// TwinCAT 3 PLC project PrensaModos
// ProgramVersion: 3.1.4023.0
// libraries:
//   Tc2_MC2, * (Beckhoff Automation GmbH)
//   Tc2_Standard, * (Beckhoff Automation GmbH)
//   Tc2_System, * (Beckhoff Automation GmbH)
//   Tc3_Module, * (Beckhoff Automation GmbH)
//   VisuDialogs, * (System)
//   VisuSymbols,3.5.10.0,System
// project tree:
//   DUTs/ estadosHome.TcDUT, EstadoMando2Manos.TcDUT, EstadosPrensa.TcDUT, Modos.TcDUT
//   / GlobalTextList.TcGTLO, PlcTask.TcTTO, Visualization Manager.TcVMO (not stored)
//   GVLs/ IO.TcGVL, VariablesGlobales.TcGVL
//   POUs/ controlejes.TcPOU, gesAlarmas.TcPOU, MAIN.TcPOU, MandoA2Mans.TcPOU, ModoAutomatico.TcPOU, resetALL.TcPOU, XestionModos.TcPOU
//   VISUs/ SimuladorPrensa.TcVIS
// real-time tasks:
//   TASK PlcTask: cycle T#10ms, priority 20, ADS port 350
// motion (NC):
//   TASK eje1 SAF: cycle T#2ms, priority 4, ADS port 501
//   TASK eje1 SVB: cycle T#10ms, priority 8, ADS port 511
//   AXIS eje1 (id 1)
//     OtherSettings: AllowMotionCmdToSlave=true
//     encoder EncType=1
//     drive DrvType=5
//       Analog: TorqueSetpointScale=10, ScaleFactorActTorque=0.1
//       TimeComp: TaskDelayCycles=1
//     controller CtrType=1
//       CtrPara: PriorControlFactor=1
//         Observer: BandWidth=20
//   AXIS Axis 2 (id 2)
//     OtherSettings: AllowMotionCmdToSlave=true
//     encoder EncType=1
//     drive DrvType=5
//       Analog: TorqueSetpointScale=10, ScaleFactorActTorque=0.1
//       TimeComp: TaskDelayCycles=1
//     controller CtrType=1
//       CtrPara: PriorControlFactor=1
//         Observer: BandWidth=20
// variable links:
//   PrensaModos/PrensaModos Instance <-> eje1 SAF/Axes/Axis 2
//     PlcTask Inputs/VariablesGlobales.eje2.NcToPlc <-> Outputs/ToPlc
//     PlcTask Outputs/VariablesGlobales.eje2.PlcToNc <-> Inputs/FromPlc
//   PrensaModos/PrensaModos Instance <-> eje1 SAF/Axes/eje1
//     PlcTask Inputs/VariablesGlobales.eje1.NcToPlc <-> Outputs/ToPlc
//     PlcTask Outputs/VariablesGlobales.eje1.PlcToNc <-> Inputs/FromPlc

CONFIGURATION PrensaModos
    RESOURCE PLC ON TwinCAT3
        TASK PlcTask(INTERVAL := T#10ms, PRIORITY := 20);
        PROGRAM MAIN WITH PlcTask : MAIN;
    END_RESOURCE
END_CONFIGURATION

// ---- DUTs/estadosHome.TcDUT
{attribute 'qualified_only'}
{attribute 'strict'}
TYPE estadosHome :
(
	subiendo:=0,
	abriendo,
	sacando,
	ok,
	espera
);
END_TYPE

// ---- DUTs/EstadoMando2Manos.TcDUT
{attribute 'qualified_only'}
{attribute 'strict'}
TYPE estadoMando2Manos:
	(
		Esperando:=0,
		Pulsado1,
		Pulsado2,
		Validado,
		Error
	);
END_TYPE

// ---- DUTs/EstadosPrensa.TcDUT
{attribute 'qualified_only'}
{attribute 'strict'}
TYPE EstadosPrensa :
(
	Parada:=0,
	Entrando,
	Pechando,
	Prensando,
	Aguantando,
	Liberando,
	Abrindo,
	Sacando
);
END_TYPE

// ---- DUTs/Modos.TcDUT
{attribute 'qualified_only'}
{attribute 'strict'}
TYPE Modos :
(
	Stop:=0,
	Auto,
	Manual,
	StopSec,
	Reseteando,
	Parando
);
END_TYPE

// ---- GVLs/IO.TcGVL
{attribute 'qualified_only'}
VAR_GLOBAL
	//Entradas modos
	Marcha AT %I*:BOOL;
	Paro AT %I*:BOOL;
	ManualAuto AT %I*:BOOL;
	SafetyOK AT %I*: BOOL;
	ResetErrores AT %I*:BOOL;
	
	//Entradas Modo Manual
	PulsadorEntrar AT %I*:BOOL;
	PulsadorSair AT %I*:BOOL;
	PulsadorPechar AT %I*:BOOL;
	PulsadorAbrir AT %I*:BOOL;
	PulsadorPrensar AT %I*:BOOL;
	PulsadorLiberar AT %I*:BOOL;
	
	//Entradas físicas mando a 2 mans
	Pulsador1 AT %I*: BOOL;
	Pulsador2 AT %I*: BOOL;
END_VAR

// ---- GVLs/VariablesGlobales.TcGVL

VAR_GLOBAL
	ModoMaquina:Modos := modos.StopSec;
	EnErro:BOOL := FALSE;
	Simular:BOOL := TRUE;
	eje1:AXIS_REF; //cinta
	eje2:AXIS_REF; //prensa
	paroAlcanzado: BOOL;
	noFallo: BOOL;
	ErrorEjes: BOOL;
	power1:BOOL:=FALSE;
	power2:BOOL:=FALSE;
	stop1:BOOL:=FALSE;
	stop2:BOOL:=FALSE;
	reset1:BOOL:=FALSE;
	reset2:BOOL:=FALSE;
	mover1:BOOL:=FALSE;
	mover2:BOOL:=FALSE;
	posicion1:UINT:=0;
	posicion2:UINT:=0;
	
END_VAR

// ---- POUs/MAIN.TcPOU
PROGRAM MAIN
VAR
END_VAR

//resetALL();
XestionModos();						//Chamada a Xestión de Modos
MandoA2Mans(LimiteSoster:=NOT modoAutomatico.goHome);	//Chamada o Mando a 2 mans
gesAlarmas();
IF mandoa2mans.Error THEN
	modoautomatico.goHome:=TRUE;
END_IF
//Se estamos en modo automático chamamos o programa
IF VariablesGlobales.ModoMaquina=modos.Auto THEN
	ModoAutomatico(bOrdenMarcha:=MandoA2Mans.Q,
	bSimular:=VariablesGlobales.Simular,
	ordenhome := io.pulsador1);	
END_IF

END_PROGRAM

// ---- POUs/XestionModos.TcPOU
PROGRAM XestionModos
VAR
	fMarcha:r_trig;
	fReset:r_trig;
	
	tResetErros:ton;
END_VAR

fMarcha(clk:=IO.marcha);
fReset(clk:=IO.ResetErrores);
power1:=TRUE;
power2:=TRUE;
stop1:=FALSE;
stop2:=FALSE;

CASE VariablesGlobales.ModoMaquina OF
	modos.Auto:
		IF IO.ManualAuto THEN
			stop1:=TRUE;
			stop2:=TRUE;
			VariablesGlobales.ModoMaquina:=modos.Manual;
		END_IF
		IF IO.Paro THEN
			VariablesGlobales.ModoMaquina:=modos.parando;
		END_IF
		IF VariablesGlobales.EnErro THEN
			VariablesGlobales.ModoMaquina:=modos.StopSec;
		END_IF
	modos.Manual:
		IF NOT IO.ManualAuto THEN
			VariablesGlobales.ModoMaquina:=modos.stop;
		END_IF
		IF VariablesGlobales.EnErro THEN
			VariablesGlobales.ModoMaquina:=modos.StopSec;
		END_IF
	
	modos.Stop:
		IF IO.ManualAuto THEN
			VariablesGlobales.ModoMaquina:=modos.Manual;
		END_IF
		IF fMarcha.q THEN
			VariablesGlobales.ModoMaquina:=modos.Auto;
		END_IF
		IF VariablesGlobales.EnErro THEN
			VariablesGlobales.ModoMaquina:=modos.StopSec;
		END_IF
	
	modos.StopSec:
		power1:=FALSE; //no tiene energía en el stopsec
		power2:=FALSE;
		IF fReset.q THEN
			VariablesGlobales.ModoMaquina:=modos.Reseteando;
			tResetErros(in:=FALSE);
		END_IF
		
	//Temos un novo modo para o reseteo, no que damos medio segundo para que, no caso de haber algunha alarma, esta salte
	modos.Reseteando:
		tResetErros(in:=TRUE, pt:=T#1S);
		IF tResetErros.Q AND NOT EnErro THEN
			VariablesGlobales.ModoMaquina:=modos.Stop;
		END_IF
		//Se o final do temporizador seguimos tendo un erro imos a modo stop seguro
		IF tResetErros.Q AND VariablesGlobales.EnErro THEN
			VariablesGlobales.ModoMaquina:=modos.StopSec;
		END_IF
	modos.Parando:
		stop1:=TRUE;
		stop2:=TRUE;
		IF paroAlcanzado THEN
			VariablesGlobales.ModoMaquina:=modos.Stop;
		END_IF
END_CASE

END_PROGRAM

// ---- POUs/MandoA2Mans.TcPOU
PROGRAM MandoA2Mans
VAR_INPUT
	LimiteSoster:BOOL;
END_VAR
VAR
	flancoP1:r_trig;
	flancoP2:r_trig;
	temp:ton;
	estadoActual:estadoMando2Manos;
END_VAR
VAR_OUTPUT
	Q:BOOL:=FALSE;
	Error:bool:=false;
END_VAR

//Valores por defecto
q:=FALSE;
Error:=FALSE;
//Control de flancos
flancoP1(clk:=IO.Pulsador1 AND ModoAutomatico.EstadoPrensa=EstadosPrensa.Parada);
flancoP2(clk:=IO.Pulsador2 AND ModoAutomatico.EstadoPrensa=EstadosPrensa.Parada);
//Temporizador para detectar a pulsación "simulatanea" dos dous pulsadores
temp(in:=estadoActual=estadoMando2Manos.Pulsado1 OR estadoActual=estadoMando2Manos.Pulsado2, pt:=T#250MS);

CASE estadoActual OF
	estadoMando2Manos.Esperando:
		IF flancoP1.Q THEN
			estadoActual:=estadoMando2Manos.Pulsado1;
		END_IF
		IF flancoP2.Q THEN
			estadoActual:=estadoMando2Manos.Pulsado2;
		END_IF
		IF flancoP1.Q AND flancoP2.Q THEN
			estadoActual:=estadoMando2Manos.Validado;
		END_IF
	estadoMando2Manos.Pulsado1:
		IF temp.Q OR NOT IO.Pulsador1 THEN
			estadoActual:=estadoMando2Manos.Esperando;
		END_IF
		IF flancoP2.Q THEN
			estadoActual:=estadoMando2Manos.Validado;
		END_IF
	estadoMando2Manos.Pulsado2:
		IF temp.Q OR NOT IO.Pulsador2 THEN
			estadoActual:=estadoMando2Manos.Esperando;
		END_IF
		IF flancoP1.Q THEN
			estadoActual:=estadoMando2Manos.Validado;
		END_IF
	estadoMando2Manos.Validado:
		q:=TRUE;
		//Se se cumplen as condicións de límite de mantemento imos a inicio
		IF LimiteSoster THEN
			estadoActual:=estadoMando2Manos.Esperando;
		END_IF
		//Se soltamos algún pulsador imos a erro
		IF NOT io.Pulsador1 OR NOT io.Pulsador2 THEN
			estadoActual:=estadoMando2Manos.Error;
		END_IF
	estadoMando2Manos.Error:
		//Erro estará a TRUE durante un ciclo
		Error:=TRUE;
		estadoActual:=estadoMando2Manos.Esperando;
END_CASE

END_PROGRAM

// ---- POUs/ModoAutomatico.TcPOU
PROGRAM ModoAutomatico
VAR_INPUT
	bOrdenMarcha: BOOL;
	bSimular:BOOL:=TRUE;
	goHome:BOOL := False;
	ordenHome:bool;
END_VAR
VAR_OUTPUT
	bFinCiclo:BOOL :=FALSE;
	EstadoPrensa: EstadosPrensa;
	estadohome: estadoshome;
	
END_VAR
VAR
	//Evolucion
	FlancoMarcha: R_trig;
	TemporizadorPrensado: Ton;
	
	//Simulacion
	TemporizadorSimulacion: TON;
	TempoSimulacion: TIME;
	ForzarErro: BOOL:=FALSE; //Esta variable permitirá forzar un erro de TimeOut
	MC_SetPosition_eje1:mc_setposition;
	MC_SetPosition_eje2:mc_setposition;
END_VAR

IF gohome THEN
	vueltacasa();
END_IF
IF NOT gohome THEN
	EvolucionEstados_Transicions();
	ActivacionActuacions_Lugares();
END_IF
IF bSimular THEN
	SimulacionAutomatico();
	simulacionejes();
END_IF

ACTION ActivacionActuacions_Lugares:
mover1:=FALSE;
mover2:=FALSE;

CASE EstadoPrensa OF
	EstadosPrensa.Entrando:
		posicion1:=1000;
		mover1:=TRUE;
	EstadosPrensa.Prensando:
		posicion2:=1000;
		mover2:=TRUE;
	EstadosPrensa.Liberando:
		posicion2:=0;
		mover2:=TRUE;
	EstadosPrensa.Sacando:
		posicion1:=0;
		mover1:=TRUE;
END_CASE
END_ACTION

ACTION EvolucionEstados_Transicions:
FlancoMarcha(clk:=bOrdenMarcha);
TemporizadorPrensado(in:=EstadoPrensa=EstadosPrensa.Aguantando, PT:=T#3S);
CASE EstadoPrensa OF
	EstadosPrensa.Parada:
		IF flancomarcha.Q THEN
			EstadoPrensa:=EstadosPrensa.Entrando;
		END_IF
	EstadosPrensa.Entrando:
		IF controlejes.MC_MoveAbsolute_eje1.Done THEN
			EstadoPrensa:=EstadosPrensa.Prensando;
		END_IF
	EstadosPrensa.Prensando:
		IF controlejes.MC_MoveAbsolute_eje2.Done THEN
			EstadoPrensa:=EstadosPrensa.Aguantando;
		END_IF
	EstadosPrensa.Aguantando:
		IF TemporizadorPrensado.Q THEN
			EstadoPrensa:=EstadosPrensa.Liberando;
		END_IF
	EstadosPrensa.Liberando:
		IF controlejes.MC_MoveAbsolute_eje1.Done THEN
			EstadoPrensa:=EstadosPrensa.Sacando;
		END_IF
	EstadosPrensa.Sacando:
		IF controlejes.MC_MoveAbsolute_eje1.Done THEN
			EstadoPrensa:=EstadosPrensa.Parada;
			bFinCiclo:=TRUE;
		END_IF
END_CASE
END_ACTION

ACTION SimulacionAutomatico:
//Se estamos simulando o pulsador1 activará ambos pulsadores
io.Pulsador2:=IO.Pulsador1;
TemporizadorSimulacion(IN:=TRUE, PT:=TempoSimulacion);
MC_SetPosition_eje1.execute:=FALSE;
MC_SetPosition_eje2.execute:=FALSE;

CASE EstadoPrensa OF
	EstadosPrensa.Parada:
		TemporizadorSimulacion(IN:=FALSE);
		TempoSimulacion:=T#5S;
		
	EstadosPrensa.Entrando:
		IF TemporizadorSimulacion.Q THEN
			MC_SetPosition_eje1.position:=1000;
			MC_SetPosition_eje1.execute:=TRUE;
			TemporizadorSimulacion(IN:=FALSE);
			TempoSimulacion:=T#2S;
		END_IF
	EstadosPrensa.Prensando:
		IF TemporizadorSimulacion.Q THEN
			MC_SetPosition_eje2.position:=1000;
			MC_SetPosition_eje2.execute:=TRUE;
			TemporizadorSimulacion(IN:=FALSE);
			TempoSimulacion:=T#3S;
		END_IF
	EstadosPrensa.Aguantando:
		TemporizadorSimulacion(IN:=FALSE);
	EstadosPrensa.Liberando:
		IF TemporizadorSimulacion.Q THEN
			MC_SetPosition_eje2.position:=0;
			MC_SetPosition_eje2.execute:=TRUE;
			TemporizadorSimulacion(IN:=FALSE);
			TempoSimulacion:=T#2S;
		END_IF
	EstadosPrensa.Sacando:
		IF TemporizadorSimulacion.Q THEN
			MC_SetPosition_eje1.position:=0;
			MC_SetPosition_eje1.execute:=TRUE;
			TemporizadorSimulacion(IN:=FALSE);
			TempoSimulacion:=T#5S;
		END_IF
END_CASE
//Se queremos forzar un erro metemoslle un minuto o temporizador
IF ForzarErro THEN
	TempoSimulacion:= T#1M;
END_IF
END_ACTION

ACTION simulacionEjes:
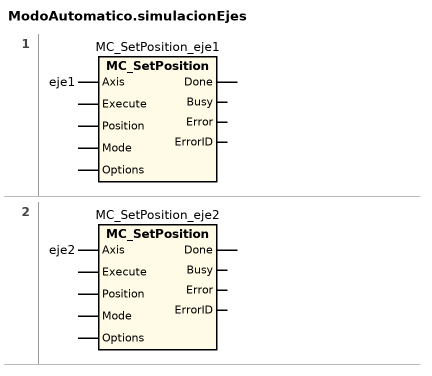
// NETWORK 1
MC_SetPosition_eje1(Axis := eje1); // MC_SetPosition

// NETWORK 2
MC_SetPosition_eje2(Axis := eje2); // MC_SetPosition
END_ACTION

ACTION vueltacasa:
mover1:=FALSE;
mover2:=FALSE;

CASE estadohome OF
	estadoshome.espera:
		IF gohome THEN
			estadohome:= estadoshome.subiendo;
		END_IF
	estadoshome.subiendo:
		posicion2:=0;
		mover2:=TRUE;
		IF controlejes.MC_MoveAbsolute_eje2.Done THEN
			estadohome:= estadoshome.sacando;
		END_IF
	estadoshome.sacando:
		posicion1:=0;
		mover1:=TRUE;
		IF controlejes.MC_MoveAbsolute_eje1.Done THEN
			estadohome:= estadoshome.ok;
		END_IF
	estadoshome.ok:
		estadohome:= estadoshome.espera;
		gohome:=FALSE;
END_CASE
END_ACTION

END_PROGRAM

// ---- POUs/controlejes.TcPOU
PROGRAM controlejes
VAR
	MC_Power_eje1: MC_Power;
	MC_Power_eje2: MC_Power;
	MC_Stop_eje1: mc_stop;
	MC_Stop_eje2: mc_stop;
	MC_Reset_eje1: mc_reset;
	MC_Reset_eje2: mc_reset;
	MC_MoveAbsolute_eje1: MC_MoveAbsolute;
	MC_MoveAbsolute_eje2: MC_MoveAbsolute;
	
	MC_ReadStatus_eje1: MC_ReadStatus;
	MC_ReadStatus_eje2: MC_ReadStatus;
	
	MC_MoveVelocity_0: MC_MoveVelocity;
END_VAR

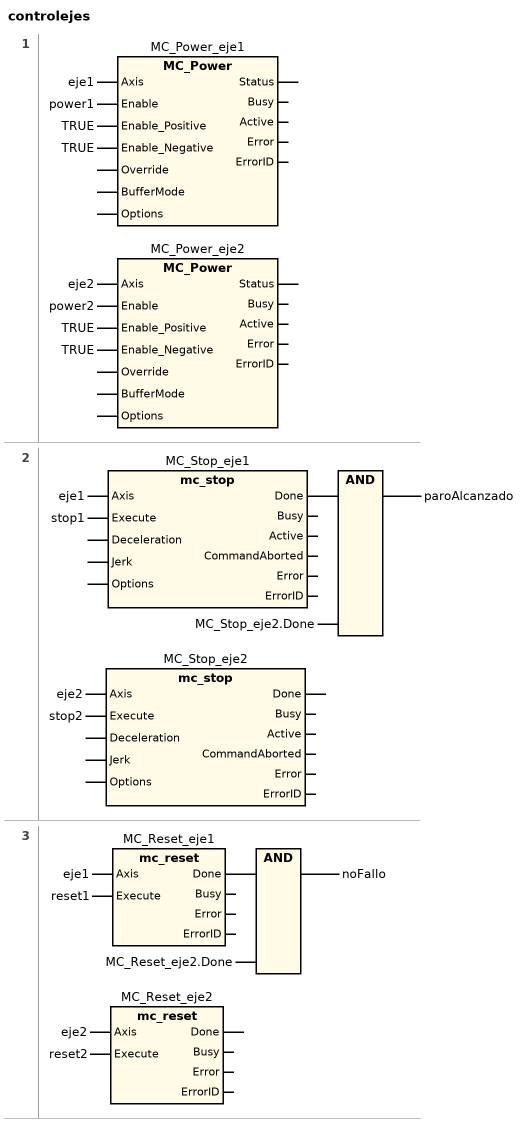
// NETWORK 1
MC_Power_eje1(Axis := eje1, Enable := power1, Enable_Positive := TRUE, Enable_Negative := TRUE); // MC_Power
MC_Power_eje2(Axis := eje2, Enable := power2, Enable_Positive := TRUE, Enable_Negative := TRUE); // MC_Power

// NETWORK 2
MC_Stop_eje1(Axis := eje1, Execute := stop1); // mc_stop
paroAlcanzado := MC_Stop_eje1.Done AND MC_Stop_eje2.Done;
MC_Stop_eje2(Axis := eje2, Execute := stop2); // mc_stop

// NETWORK 3
MC_Reset_eje1(Axis := eje1, Execute := reset1); // mc_reset
noFallo := MC_Reset_eje1.Done AND MC_Reset_eje2.Done;
MC_Reset_eje2(Axis := eje2, Execute := reset2); // mc_reset

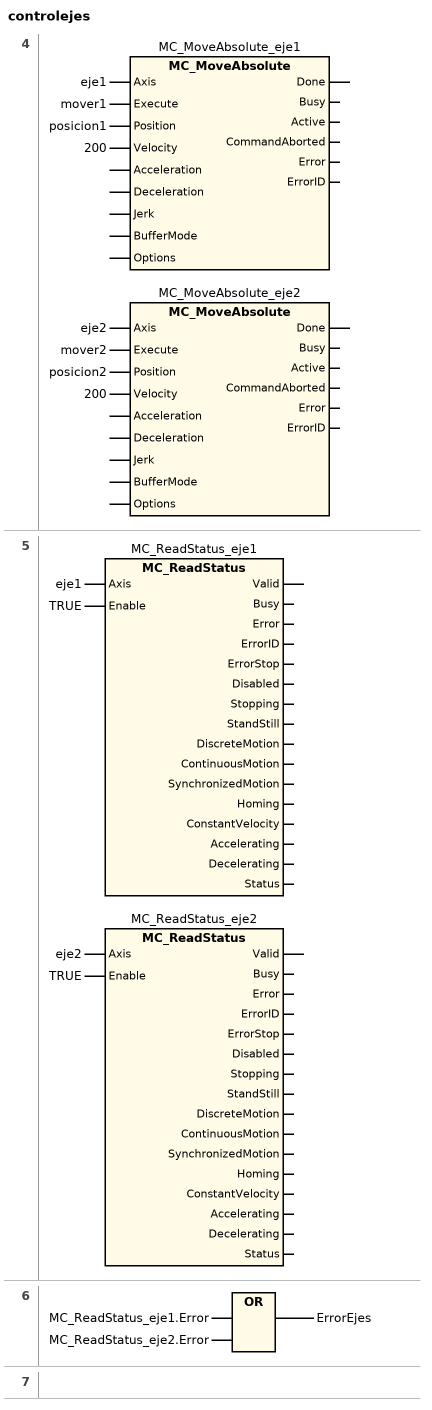
// NETWORK 4
MC_MoveAbsolute_eje1(Axis := eje1, Execute := mover1, Position := posicion1, Velocity := 200); // MC_MoveAbsolute
MC_MoveAbsolute_eje2(Axis := eje2, Execute := mover2, Position := posicion2, Velocity := 200); // MC_MoveAbsolute

// NETWORK 5
MC_ReadStatus_eje1(Axis := eje1, Enable := TRUE); // MC_ReadStatus
MC_ReadStatus_eje2(Axis := eje2, Enable := TRUE); // MC_ReadStatus

// NETWORK 6
ErrorEjes := MC_ReadStatus_eje1.Error OR MC_ReadStatus_eje2.Error;

// NETWORK 7

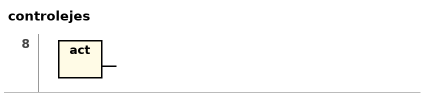
// NETWORK 8
act();

ACTION ACT:
// NETWORK 1
END_ACTION

ACTION ACT_1:
// NETWORK 1
END_ACTION

END_PROGRAM

// ---- POUs/gesAlarmas.TcPOU
PROGRAM gesAlarmas
VAR
	TempTimeOUT:ton;
	EstAnt:EstadosPrensa;
	
	PrimeiroErro:INT;
	Erros:ARRAY[1..9] OF BOOL;
	contador:INT;

END_VAR

IF Variablesglobales.ModoMaquina=modos.Reseteando THEN
	primeiroerro:=0;
	FOR contador:=1 TO 9 DO
		erros[contador]:=FALSE;
	END_FOR
END_IF

temptimeout(in:=estant=modoautomatico.EstadoPrensa AND 
	variablesglobales.ModoMaquina = modos.Auto AND 
	modoautomatico.estadoprensa <> estadosprensa.Parada, pt:=T#15S); //la vaina esta <> es un distinto
IF tempTimeout.q THEN 
	erros[1]:=TRUE;
	IF primeiroErro=0 THEN
		primeiroErro:=1;
	END_IF
END_IF

//error ejes
IF ErrorEjes THEN
	erros[2]:=TRUE;
	IF primeiroerro=0 THEN
		primeiroerro:=2;
	END_IF
END_IF

//seta emergency
IF NOT io.SafetyOK THEN
	erros[3]:=TRUE;
	IF primeiroerro=0 THEN
		primeiroerro:=3;
	END_IF	
END_IF

//mando dos manos
IF mandoa2mans.Error THEN
	erros[4]:=TRUE;
	IF primeiroerro=0 THEN
		primeiroerro:=4;
	END_IF	
END_IF

VariablesGlobales.EnErro := PrimeiroErro<>0;
estant:=modoautomatico.EstadoPrensa;

END_PROGRAM

// ---- POUs/resetALL.TcPOU
PROGRAM resetALL
VAR
END_VAR

IO.ElectroEntrar:=FALSE;
IO.ElectroPechar:=FALSE;
IO.ElectroPrensar:=FALSE;
IO.ElectroLiberar:=FALSE;
IO.ElectroAbrir:=FALSE;
IO.ElectroSair:=FALSE;

END_PROGRAM

// ---- GlobalTextList.TcGTLO
TEXTLIST GlobalTextList
  44 = 'ALARMAS ACTIVAS'
  713 = 'capasao %s'
  221 = 'Estado: %s'
  844 = 'FORZAR TIMEOUT'
  623 = 'Manual \tAutomático'
  656 = 'Marcha'
  640 = 'Modo %s'
  282 = 'nº error %s'
  165 = 'Paro'
  101 = 'Primeiro erro %s'
  364 = 'Pulsador'
  983 = 'Pulsador1'
  683 = 'Pulsador2'
  773 = 'Rearme'
  75 = 'Simular'
END_TEXTLIST

// ---- VISUs/SimuladorPrensa.TcVIS
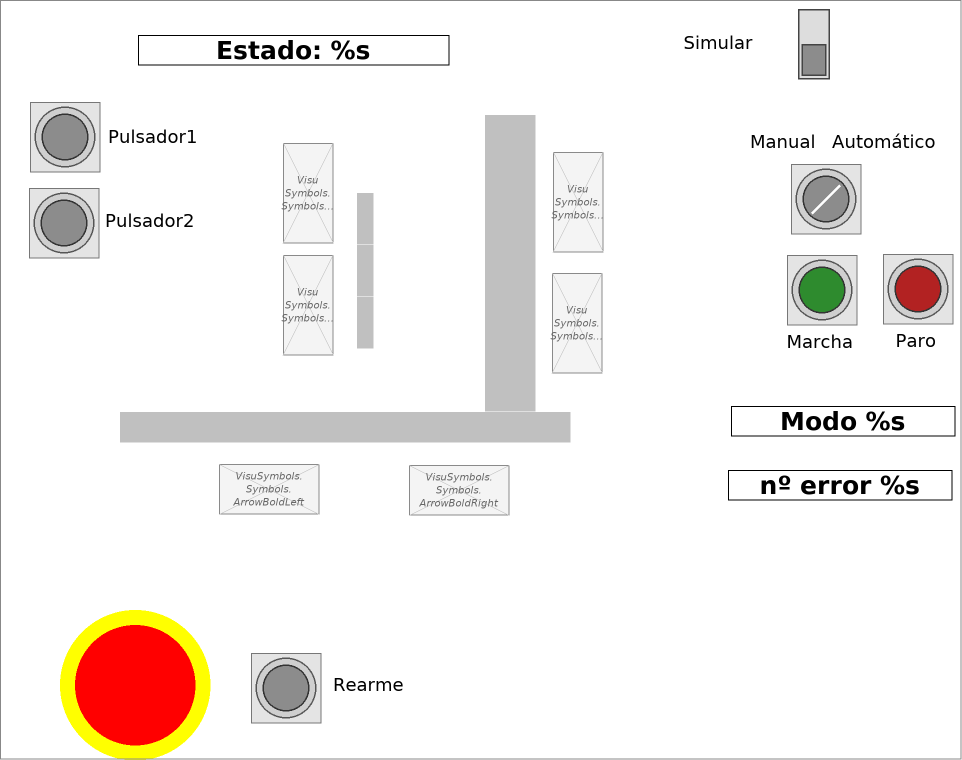
VISUALIZATION SimuladorPrensa  // 962x760
    PushSwitch (30,102 70x70), variable: IO.Pulsador1, behaviour: TAP, style: Switch-PushSwitch-Gray
    Rectangle (120,412 150x30), colour toggle: IO.SensorFora
        OnMouseClick: toggle IO.SensorFora
    Rectangle (270,412 150x30), colour toggle: Not IO.SensorFora and Not io.SensorDentro
    Rectangle (420,412 150x30), colour toggle: IO.SensorDentro
        OnMouseClick: toggle IO.SensorDentro
    Rectangle (357,193 16x51), colour toggle: IO.SensorAberto
        OnMouseClick: toggle IO.SensorAberto
    Rectangle (357,245 16x51), colour toggle: Not IO.SensorAberto and Not IO.SensorPechado
    Rectangle (357,297 16x51), colour toggle: IO.SensorPechado
        OnMouseClick: toggle IO.SensorPechado
    Rectangle (485,115 50x100), colour toggle: IO.SensorArriba
        OnMouseClick: toggle IO.SensorArriba
    Rectangle (485,214 50x100), colour toggle: Not io.SensorArriba and Not IO.SensorAbaixo
    Rectangle (485,311 50x100), colour toggle: IO.SensorAbaixo
        OnMouseClick: toggle IO.SensorAbaixo
    Rectangle (138,35 311x30), "Estado: %s", text variable: ModoAutomatico.EstadoPrensa
    Image (283,143 50x100), colour toggle: IO.ElectroAbrir, image: VisuSymbols.Symbols.ArrowBoldUp
        OnMouseDown: toggle IO.PulsadorAbrir
        OnMouseUp: toggle IO.PulsadorAbrir
    Image (283,255 50x100), colour toggle: IO.ElectroPechar, image: VisuSymbols.Symbols.ArrowBoldDown
        OnMouseDown: toggle IO.PulsadorPechar
        OnMouseUp: toggle IO.PulsadorPechar
    Image (553,152 50x100), colour toggle: IO.ElectroLiberar, image: VisuSymbols.Symbols.ArrowBoldUp
        OnMouseDown: toggle IO.PulsadorLiberar
        OnMouseUp: toggle IO.PulsadorLiberar
    Image (552,273 50x100), colour toggle: IO.ElectroPrensar, image: VisuSymbols.Symbols.ArrowBoldDown
        OnMouseDown: toggle IO.PulsadorPrensar
        OnMouseUp: toggle IO.PulsadorPrensar
    Image (409,465 100x50), colour toggle: IO.ElectroEntrar, image: VisuSymbols.Symbols.ArrowBoldRight
        OnMouseDown: toggle IO.PulsadorEntrar
        OnMouseUp: toggle IO.PulsadorEntrar
    Image (219,464 100x50), colour toggle: IO.ElectroSair, image: VisuSymbols.Symbols.ArrowBoldLeft
        OnMouseDown: toggle IO.PulsadorSair
        OnMouseUp: toggle IO.PulsadorSair
    Ellipse (60,610 150x150)
    Ellipse (75,625 120x120), colour toggle: Not IO.SafetyOK
        OnMouseClick: toggle IO.SafetyOK
    PushSwitch (251,653 70x70), variable: IO.ResetErrores, behaviour: TAP, style: Switch-PushSwitch-Gray
    RotarySwitch (791,164 70x70), variable: IO.ManualAuto, behaviour: TOGGLE, style: Switch-RotarySwitch-Gray
    PushSwitch (787,255 70x70), variable: IO.Marcha, behaviour: TAP, style: Switch-PushSwitch-Green
    Rectangle (731,406 224x30), "Modo %s", text variable: VariablesGlobales.ModoMaquina
    PushSwitch (883,254 70x70), variable: IO.Paro, behaviour: TOGGLE, style: Switch-PushSwitch-Red
    Label (327,663 83x44), "Rearme"
    Label (107,115 92x44), "Pulsador1"
    Label (741,120 204x44), "Manual Automático"
    Label (774,320 92x44), "Marcha"
    Label (870,319 92x44), "Paro"
    PushSwitch (29,188 70x70), variable: IO.Pulsador2, behaviour: TAP, style: Switch-PushSwitch-Gray
    Label (104,199 92x44), "Pulsador2"
    DipSwitch (779,9 70x70), variable: VariablesGlobales.Simular, behaviour: TOGGLE, style: Switch-DipSwitch-Gray
    Label (672,21 92x44), "Simular"
    Rectangle (728,470 224x30), "nº error %s", text variable: gesAlarmas.PrimeiroErro
END_VISUALIZATION
